FUNCTION_BLOCK AX_SPLIT3 (* SPLIT 1 AX into 3 AX *)
  (* Standard: 61499-2; Description: Copyright (c) 2025 HR Agrartechnik GmbH This program and the accompanying materials are made available under the terms of the Eclipse Public License 2.0 which is available at https://www.eclipse.org/legal/epl-2.0/ SPDX-License-Identifier: EPL-2.0 *)
  (* Version 1.0, 2025-01-24, Franz Höpfinger, HR Agrartechnik GmbH *)
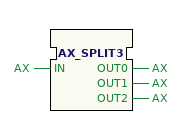
  SOCKETS
    IN : AX;
  END_SOCKETS
  PLUGS
    OUT0 : AX;
    OUT1 : AX;
    OUT2 : AX;
  END_PLUGS
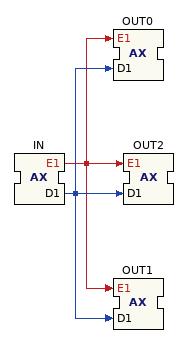
  EVENT_CONNECTIONS
    IN.E1 TO OUT0.E1;
    IN.E1 TO OUT1.E1;
    IN.E1 TO OUT2.E1;
  END_CONNECTIONS
  DATA_CONNECTIONS
    IN.D1 TO OUT0.D1;
    IN.D1 TO OUT1.D1;
    IN.D1 TO OUT2.D1;
  END_CONNECTIONS
END_FUNCTION_BLOCK
